{attribute 'linkalways'} 
{attribute 'no_explicit_call' := 'This FB is a CLASS and must be accessed using methods or properties'}
{attribute 'enable_dynamic_creation'}
FUNCTION_BLOCK StopCommand EXTENDS AxisCommand
VAR
	_deceleration : LREAL;
	_jerk : LREAL;
END_VAR

METHOD FB_init : BOOL
VAR_INPUT
	bInitRetains : BOOL; // if TRUE, the retain variables are initialized (warm start / cold start)
	bInCopyCode : BOOL;  // if TRUE, the instance afterwards gets moved into the copy code (online change)
	axisRef : REFERENCE TO Axis;
END_VAR
_axisRef REF= axisRef;
END_METHOD

METHOD PROTECTED WhileBusy
VAR_INPUT
	CommandState : I_CommandBusyState;
END_VAR
VAR_INST
	_fb : MC_Stop;
END_VAR
_fb(
	Axis := _axisRef._InternalAxisRef,
	Execute := TRUE,
	Deceleration := _deceleration,
	Jerk := _jerk
);

IF NOT _fb.Done THEN
	RETURN;
END_IF

_fb(Axis := _axisRef._InternalAxisRef, Execute := FALSE);
CommandState.SetDone();
END_METHOD

END_FUNCTION_BLOCK

(* stored: Version 1.1.0.1, ProductVersion 3.1.4024.12
   POU StopCommand: Id {5aedb90c-1a45-4333-8ff4-9287e637597f}, SpecialFunc None
   Folder Constructor: Id {dc0acbb8-17a6-426e-9fbb-199eb0e53e8a}
   Method FB_init: Id {08dabbdf-6250-4037-ba02-16e1df44f728}
   Method WhileBusy: Id {0538c416-e656-406a-91d4-185131119da4} *)
